SYSTEM test_CLIENT_SERVER
  (* Version 1.0, 2023-10-23, franz *)
  PACKAGE Training_CLIENT_SERVER;
  IMPORT VV::const::Computers::myComputers;
  IMPORT VV::const::Computers::myComputers::C_PC_CLIENT;
  IMPORT VV::const::Computers::myComputers::C_PC_SERVER;
  IMPORT VV::const::ports::myPorts;
  IMPORT VV::const::ports::myPorts::PORT_A0;
  IMPORT VV::const::ports::myPorts::PORT_A1;
  IMPORT VV::const::ports::myPorts::PORT_A2;
  IMPORT VV::const::ports::myPorts::PORT_A3;
  IMPORT VV::const::ports::myPorts::PORT_B0;
  IMPORT VV::const::ports::myPorts::PORT_B1;
  IMPORT VV::const::ports::myPorts::PORT_B2;
  IMPORT VV::const::ports::myPorts::PORT_B3;
  IMPORT logiBUS::io::DI::logiBUS_DI::Input_I1;
  IMPORT logiBUS::io::DI::logiBUS_DI::Input_I2;
  IMPORT logiBUS::io::DI::logiBUS_DI::Input_I3;
  IMPORT logiBUS::io::DI::logiBUS_DI::Input_I4;
  IMPORT logiBUS::io::DO_LED::LED_COLOURS;
  IMPORT logiBUS::io::DO_LED::LED_COLOURS::LED_BLUE;
  IMPORT logiBUS::io::DO_LED::LED_COLOURS::LED_GREEN;
  IMPORT logiBUS::io::DO_LED::LED_COLOURS::LED_RED;
  IMPORT logiBUS::io::DO_LED::LED_COLOURS::LED_YELLOW;
  IMPORT logiBUS::io::DO_LED::LED_FREQ;
  IMPORT logiBUS::io::DO_LED::LED_FREQ::LED_5HZ;
  IMPORT logiBUS::io::DO_LED::LED_strip;
  IMPORT logiBUS::io::DO_LED::LED_strip::Output_strip;
  APPLICATION App_CLIENT_SERVER
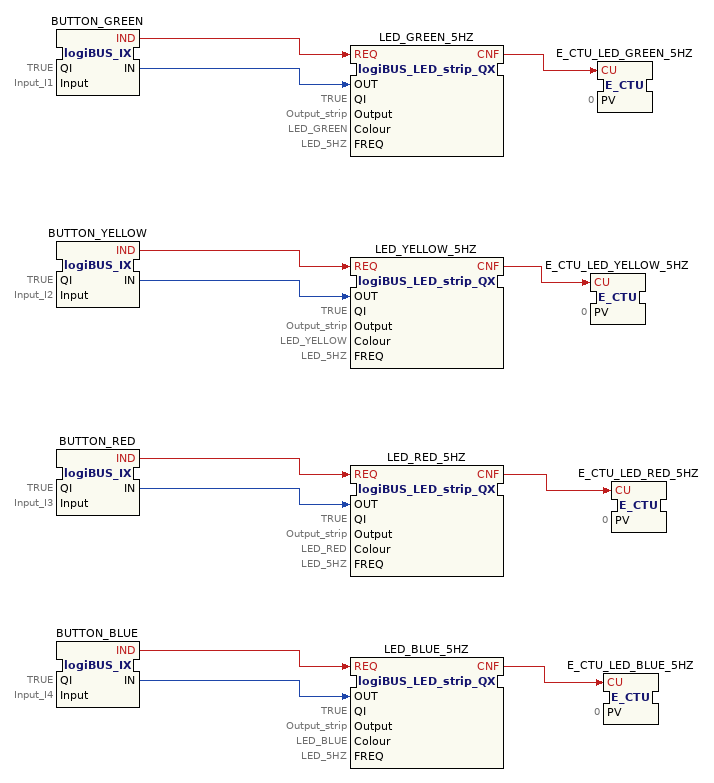
    FBS
      BUTTON_RED : logiBUS::io::DI::logiBUS_IX(QI := TRUE, Input := Input_I3);
      BUTTON_YELLOW : logiBUS::io::DI::logiBUS_IX(QI := TRUE, Input := Input_I2);
      BUTTON_BLUE : logiBUS::io::DI::logiBUS_IX(QI := TRUE, Input := Input_I4);
      LED_YELLOW_5HZ : logiBUS::io::DO_LED::logiBUS_LED_strip_QX(QI := TRUE, Output := Output_strip, Colour := LED_YELLOW, FREQ := LED_5HZ);
      LED_BLUE_5HZ : logiBUS::io::DO_LED::logiBUS_LED_strip_QX(QI := TRUE, Output := Output_strip, Colour := LED_BLUE, FREQ := LED_5HZ);
      LED_RED_5HZ : logiBUS::io::DO_LED::logiBUS_LED_strip_QX(QI := TRUE, Output := Output_strip, Colour := LED_RED, FREQ := LED_5HZ);
      BUTTON_GREEN : logiBUS::io::DI::logiBUS_IX(QI := TRUE, Input := Input_I1);
      LED_GREEN_5HZ : logiBUS::io::DO_LED::logiBUS_LED_strip_QX(QI := TRUE, Output := Output_strip, Colour := LED_GREEN, FREQ := LED_5HZ);
      E_CTU_LED_GREEN_5HZ : iec61499::events::E_CTU(PV := 0);
      E_CTU_LED_YELLOW_5HZ : iec61499::events::E_CTU(PV := 0);
      E_CTU_LED_RED_5HZ : iec61499::events::E_CTU(PV := 0);
      E_CTU_LED_BLUE_5HZ : iec61499::events::E_CTU(PV := 0);
    END_FBS
    EVENT_CONNECTIONS
      BUTTON_RED.IND TO LED_RED_5HZ.REQ;
      BUTTON_YELLOW.IND TO LED_YELLOW_5HZ.REQ;
      BUTTON_BLUE.IND TO LED_BLUE_5HZ.REQ;
      BUTTON_GREEN.IND TO LED_GREEN_5HZ.REQ;
      LED_GREEN_5HZ.CNF TO E_CTU_LED_GREEN_5HZ.CU;
      LED_YELLOW_5HZ.CNF TO E_CTU_LED_YELLOW_5HZ.CU;
      LED_RED_5HZ.CNF TO E_CTU_LED_RED_5HZ.CU;
      LED_BLUE_5HZ.CNF TO E_CTU_LED_BLUE_5HZ.CU;
    END_CONNECTIONS
    DATA_CONNECTIONS
      BUTTON_RED.IN TO LED_RED_5HZ.OUT;
      BUTTON_YELLOW.IN TO LED_YELLOW_5HZ.OUT;
      BUTTON_BLUE.IN TO LED_BLUE_5HZ.OUT;
      BUTTON_GREEN.IN TO LED_GREEN_5HZ.OUT;
    END_CONNECTIONS
  END_APPLICATION
  DEVICE FORTE_PC_CLIENT : iec61499::system::FORTE_PC(MGR_ID := C_PC_SERVER (* Device manager socket ID *))
    {SET_ATTRIBUTE(Profile, HOLOBLOC)}
    RESOURCE EMB_RES_CLIENT : iec61499::system::EMB_RES
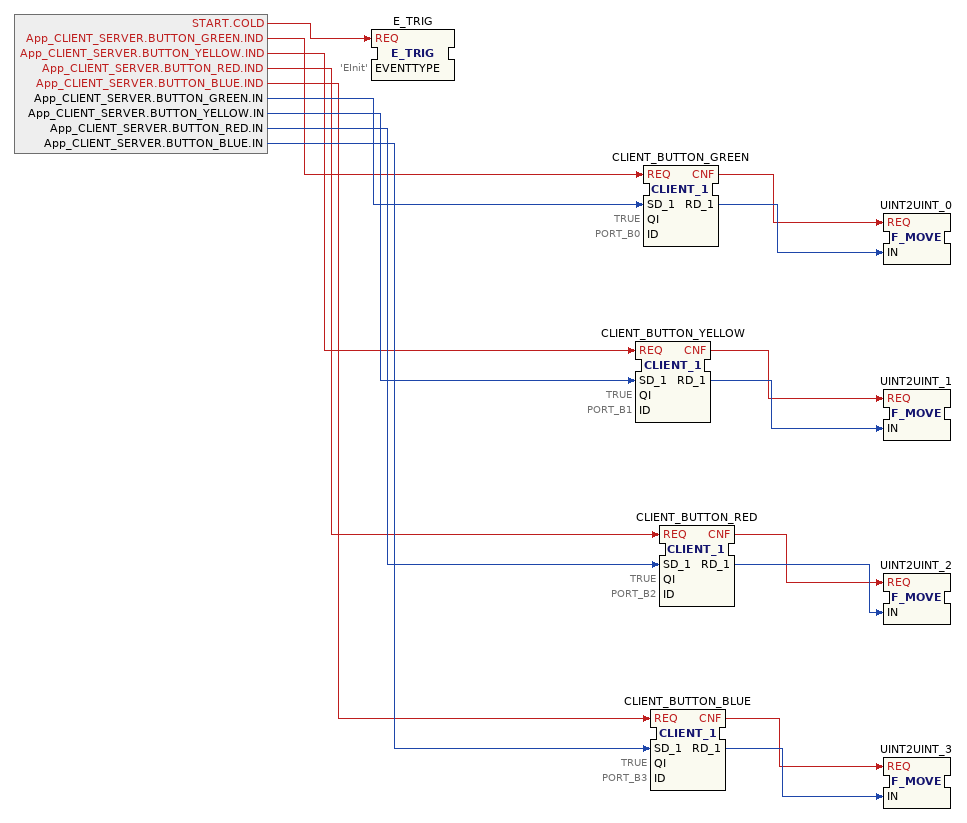
      FBS
        CLIENT_BUTTON_GREEN : iec61499::net::CLIENT_1(QI := TRUE, ID := PORT_B0);
        CLIENT_BUTTON_YELLOW : iec61499::net::CLIENT_1(QI := TRUE, ID := PORT_B1);
        CLIENT_BUTTON_RED : iec61499::net::CLIENT_1(QI := TRUE, ID := PORT_B2);
        CLIENT_BUTTON_BLUE : iec61499::net::CLIENT_1(QI := TRUE, ID := PORT_B3);
        UINT2UINT_0 : iec61131::selection::F_MOVE; {SET_ATTRIBUTE(DataType, UINT)}
        UINT2UINT_1 : iec61131::selection::F_MOVE; {SET_ATTRIBUTE(DataType, UINT)}
        UINT2UINT_2 : iec61131::selection::F_MOVE; {SET_ATTRIBUTE(DataType, UINT)}
        UINT2UINT_3 : iec61131::selection::F_MOVE; {SET_ATTRIBUTE(DataType, UINT)}
        E_TRIG : iec61499::events::E_TRIG(EVENTTYPE := 'EInit');
      END_FBS
      EVENT_CONNECTIONS
        CLIENT_BUTTON_GREEN.CNF TO UINT2UINT_0.REQ;
        CLIENT_BUTTON_RED.CNF TO UINT2UINT_2.REQ;
        CLIENT_BUTTON_YELLOW.CNF TO UINT2UINT_1.REQ;
        CLIENT_BUTTON_BLUE.CNF TO UINT2UINT_3.REQ;
        START.COLD TO E_TRIG.REQ;
        App_CLIENT_SERVER.BUTTON_GREEN.IND TO CLIENT_BUTTON_GREEN.REQ;
        App_CLIENT_SERVER.BUTTON_YELLOW.IND TO CLIENT_BUTTON_YELLOW.REQ;
        App_CLIENT_SERVER.BUTTON_RED.IND TO CLIENT_BUTTON_RED.REQ;
        App_CLIENT_SERVER.BUTTON_BLUE.IND TO CLIENT_BUTTON_BLUE.REQ;
      END_CONNECTIONS
      DATA_CONNECTIONS
        CLIENT_BUTTON_GREEN.RD_1 TO UINT2UINT_0.IN;
        CLIENT_BUTTON_RED.RD_1 TO UINT2UINT_2.IN;
        CLIENT_BUTTON_YELLOW.RD_1 TO UINT2UINT_1.IN;
        CLIENT_BUTTON_BLUE.RD_1 TO UINT2UINT_3.IN;
        App_CLIENT_SERVER.BUTTON_GREEN.IN TO CLIENT_BUTTON_GREEN.SD_1;
        App_CLIENT_SERVER.BUTTON_YELLOW.IN TO CLIENT_BUTTON_YELLOW.SD_1;
        App_CLIENT_SERVER.BUTTON_RED.IN TO CLIENT_BUTTON_RED.SD_1;
        App_CLIENT_SERVER.BUTTON_BLUE.IN TO CLIENT_BUTTON_BLUE.SD_1;
      END_CONNECTIONS
    END_RESOURCE
  END_DEVICE
  DEVICE FORTE_PC_SERVER : iec61499::system::FORTE_PC(MGR_ID := C_PC_CLIENT (* Device manager socket ID *))
    {SET_ATTRIBUTE(Profile, HOLOBLOC)}
    RESOURCE EMB_RES_SERVER : iec61499::system::EMB_RES
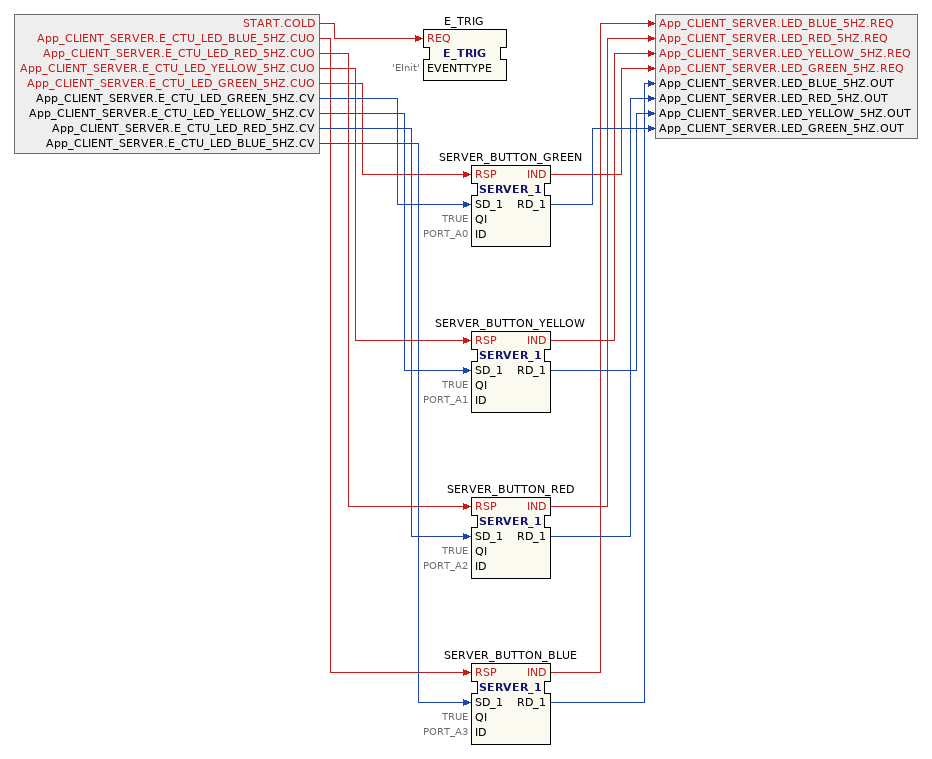
      FBS
        SERVER_BUTTON_GREEN : iec61499::net::SERVER_1(QI := TRUE, ID := PORT_A0);
        SERVER_BUTTON_RED : iec61499::net::SERVER_1(QI := TRUE, ID := PORT_A2);
        SERVER_BUTTON_YELLOW : iec61499::net::SERVER_1(QI := TRUE, ID := PORT_A1);
        SERVER_BUTTON_BLUE : iec61499::net::SERVER_1(QI := TRUE, ID := PORT_A3);
        E_TRIG : iec61499::events::E_TRIG(EVENTTYPE := 'EInit');
      END_FBS
      EVENT_CONNECTIONS
        START.COLD TO E_TRIG.REQ;
        App_CLIENT_SERVER.E_CTU_LED_BLUE_5HZ.CUO TO SERVER_BUTTON_BLUE.RSP;
        App_CLIENT_SERVER.E_CTU_LED_RED_5HZ.CUO TO SERVER_BUTTON_RED.RSP;
        App_CLIENT_SERVER.E_CTU_LED_YELLOW_5HZ.CUO TO SERVER_BUTTON_YELLOW.RSP;
        App_CLIENT_SERVER.E_CTU_LED_GREEN_5HZ.CUO TO SERVER_BUTTON_GREEN.RSP;
        SERVER_BUTTON_BLUE.IND TO App_CLIENT_SERVER.LED_BLUE_5HZ.REQ;
        SERVER_BUTTON_RED.IND TO App_CLIENT_SERVER.LED_RED_5HZ.REQ;
        SERVER_BUTTON_YELLOW.IND TO App_CLIENT_SERVER.LED_YELLOW_5HZ.REQ;
        SERVER_BUTTON_GREEN.IND TO App_CLIENT_SERVER.LED_GREEN_5HZ.REQ;
      END_CONNECTIONS
      DATA_CONNECTIONS
        App_CLIENT_SERVER.E_CTU_LED_GREEN_5HZ.CV TO SERVER_BUTTON_GREEN.SD_1;
        App_CLIENT_SERVER.E_CTU_LED_YELLOW_5HZ.CV TO SERVER_BUTTON_YELLOW.SD_1;
        App_CLIENT_SERVER.E_CTU_LED_RED_5HZ.CV TO SERVER_BUTTON_RED.SD_1;
        App_CLIENT_SERVER.E_CTU_LED_BLUE_5HZ.CV TO SERVER_BUTTON_BLUE.SD_1;
        SERVER_BUTTON_BLUE.RD_1 TO App_CLIENT_SERVER.LED_BLUE_5HZ.OUT;
        SERVER_BUTTON_RED.RD_1 TO App_CLIENT_SERVER.LED_RED_5HZ.OUT;
        SERVER_BUTTON_YELLOW.RD_1 TO App_CLIENT_SERVER.LED_YELLOW_5HZ.OUT;
        SERVER_BUTTON_GREEN.RD_1 TO App_CLIENT_SERVER.LED_GREEN_5HZ.OUT;
      END_CONNECTIONS
    END_RESOURCE
  END_DEVICE
  MAPPINGS
    App_CLIENT_SERVER.BUTTON_BLUE ON FORTE_PC_CLIENT.EMB_RES_CLIENT;
    App_CLIENT_SERVER.BUTTON_RED ON FORTE_PC_CLIENT.EMB_RES_CLIENT;
    App_CLIENT_SERVER.BUTTON_YELLOW ON FORTE_PC_CLIENT.EMB_RES_CLIENT;
    App_CLIENT_SERVER.LED_RED_5HZ ON FORTE_PC_SERVER.EMB_RES_SERVER;
    App_CLIENT_SERVER.LED_YELLOW_5HZ ON FORTE_PC_SERVER.EMB_RES_SERVER;
    App_CLIENT_SERVER.LED_BLUE_5HZ ON FORTE_PC_SERVER.EMB_RES_SERVER;
    App_CLIENT_SERVER.LED_GREEN_5HZ ON FORTE_PC_SERVER.EMB_RES_SERVER;
    App_CLIENT_SERVER.BUTTON_GREEN ON FORTE_PC_CLIENT.EMB_RES_CLIENT;
    App_CLIENT_SERVER.E_CTU_LED_YELLOW_5HZ ON FORTE_PC_SERVER.EMB_RES_SERVER;
    App_CLIENT_SERVER.E_CTU_LED_RED_5HZ ON FORTE_PC_SERVER.EMB_RES_SERVER;
    App_CLIENT_SERVER.E_CTU_LED_GREEN_5HZ ON FORTE_PC_SERVER.EMB_RES_SERVER;
    App_CLIENT_SERVER.E_CTU_LED_BLUE_5HZ ON FORTE_PC_SERVER.EMB_RES_SERVER;
  END_MAPPINGS
END_SYSTEM
